{attribute 'qualified_only'}
{attribute 'strict'}
TYPE E_CmdResult :
(
    eBusy  := 0,   // command still running, keep calling it
    eDone  := 1,   // command finished successfully -> advance the step
    eError := 2    // command failed (e.g. move timeout) -> handle the error
) DINT;
END_TYPE

(* stored: Version 1.1.0.1
   DUT E_CmdResult: Id {4a7d9ed1-2ff3-4cd0-8ad8-f2a7fa8c367e} *)
